{attribute 'qualified_only'}
{attribute 'strict'}
TYPE States :
(
	Init := 0,
	Idle,
	MoveToPickUp,
	PickUpDown,
	PickUpUp,
	MoveX,
	MoveY,
	DropDown,
	DropUp,
	PalletFull
);
END_TYPE

(* stored: Version 1.1.0.1, ProductVersion 3.1.4022.12
   DUT States: Id {27b41ea7-0afd-4559-8ac7-01b9f3b8d6f2} *)
